// TIA Portal V17 export
// export: Created 2025-03-05T08:03:34.1256908Z, ExportSetting WithDefaults, DisplayName Totally Integrated Automation Portal, DisplayVersion V17 Update 8, DisplayName TIA Portal Openness, DisplayVersion V17 Update 8, DisplayName TIA Portal Version Control Interface, DisplayVersion V17, DisplayName SINAMICS Startdrive Advanced, DisplayVersion V17 SP2, DisplayName SINAMICS Startdrive G110M, G120, G120C, G120D, G120P, G115D, DisplayVersion V17 SP2, DisplayName SINAMICS Startdrive G130, G150, S120, S150, SINAMICS MV, S210, DisplayVersion V17 SP2, DisplayName STEP 7 Professional, DisplayVersion V17 Update 8, DisplayName SINUMERIK ONE STEP 7 Toolbox, DisplayVersion V17 Update 12, DisplayName SINUMERIK 840D sl STEP 7 Toolbox, DisplayVersion V17 Update 12, DisplayName STEP 7 Safety, DisplayVersion V17 Update 6, DisplayName WinCC Advanced, DisplayVersion V17 Update 8
DATA_BLOCK "DB22741_LOAD_FEEDER_TIME_SEQUENCE_HOPPER_3_UNIT_02"   // DB22741
{ DB_Accessible_From_OPC_UA := 'FALSE' }
VERSION : 0.1
// stored: AutoNumber false, DBAccessibleFromOPCUA false, DBAccessibleFromWebserver true, InstanceOfName FB22701_LOAD_FEEDER_SEQUENCE_TIME, InstanceOfType FB
"FB22701_LOAD_FEEDER_SEQUENCE_TIME"
   // VAR_INPUT
   //    iCONTROL_ON_DELAYED : Bool;
   //    iPNEUMATIC_FEEDBACK_ON : Bool;
   //    iFEEDER_PROFINET_MODE_ACTIVE_FAULT : Bool;
   //    iFEEDER_LINE_NOT_READY_FAULT : Bool;
   //    iMOTOR_STIRRER_CONDITIONS : Bool;
   //    iHOPPER_FEEDBACK_PRESSURE : Real;
   //    iHOPPER_MOTOR_STIRRER_FEEDBACK_SPEED : Real;
   //    iPOWDER_FEEDER_HOPPER_FEEDBACK_PRESSURE : Real;
   //    iTRANSFER_POWDER_VALVE_FEEDBACK_ON : Bool;
   //    iTRANSFER_POWDER_VALVE_FEEDBACK_OFF : Bool;
   //    iPOWDER_FLOW_ON : Bool;
   //    iSTART_MANUAL_REQUEST : Bool;
   //    iSTART_SEMI_REQUEST : Bool;
   //    iSTART_AUTO_REQUEST : Bool;
   //    iSTOP_MANUAL_REQUEST : Bool;
   //    iSTOP_SEMI_REQUEST : Bool;
   //    iSTOP_AUTO_REQUEST : Bool;
   // END_VAR
   // VAR_OUTPUT
   //    oEXCEEDED_TIME_ALARM : Bool;
   //    oOUT_OF_RANGE_ALARM : Bool;
   //    oLOST_CONDITIONS : Bool;
   //    oIS_ALARMS : Bool;
   // END_VAR
   // VAR_IN_OUT
   //    MOTOR_STIRRER_SETPOINT : DInt;
   //    PRESSURE_SETPOINT : Real;
   // END_VAR
   // VAR RETAIN
   //    DATA_SEQUENCE : "GENERAL_DATA_SEQUENCES";
   //    HMI_STANDARD : "HMI_DATA_START_STOP";
   //    INPUT_SETTINGS : Struct
   //       UNIT_NUMBER : Int := 2;
   //       HOPPER_NUMBER : Int := 3;
   //    END_STRUCT;
   //    HMI_SEQUENCE : Struct
   //       HMI_SEQUENCE_RUNNING : Bool;
   //       HMI_SEQUENCE_DONE : Bool;
   //       HMI_SET_TIME_LOAD : UDInt;
   //       HMI_MAX_ON_SET_TIME : UDInt;
   //       HMI_FEEDBACK_TIME_LOAD : Int;
   //       HMI_PRESSURE_INCREMENT : Real;
   //    END_STRUCT;
   //    ACTIONS_SEQUENCE : Struct
   //       REQ_START_TRANSFER_POWDER_VALVE : Bool;
   //       REQ_STOP_TRANSFER_POWDER_VALVE : Bool;
   //       REQ_START_PRESSURE_GAS_CONTROL : Bool;
   //       REQ_STOP_PRESSURE_GAS_CONTROL : Bool;
   //       REQ_START_PRESSURE_GAS_VALVE : Bool;
   //       REQ_STOP_PRESSURE_GAS_VALVE : Bool;
   //       REQ_START_RELIEF_GAS_VALVE : Bool;
   //       REQ_STOP_RELIEF_GAS_VALVE : Bool;
   //       SETPOINT_PRESSURE : Real;
   //       REQUEST_START_MOTOR_STIRRER : Bool;
   //       REQUEST_STOP_MOTOR_STIRRER : Bool;
   //       SETPOINT_MOTOR_STIRRER : DInt;
   //    END_STRUCT;
   //    CONTROL_SEQUENCE : Struct
   //       HOPPER_PRESSURE_IN_RANGE : Bool;
   //       HOPPER_MOTOR_STIRRER_IN_RANGE : Bool;
   //       HOPPER_STIRRER_LOW_RANGE : DInt;
   //       HOPPER_STIRRER_HIGH_RANGE : DInt;
   //       HOPPER_PRESSURE_LOW_RANGE : Real;
   //       HOPPER_PRESSURE_HIGH_RANGE : Real;
   //       HOPPER_PRESSURE_INCREMENT : Real;
   //       TIMER_IS_OVER : Bool;
   //       INITIAL_TIME_SET : DInt;
   //       TIMER_MATERIAL_APPLIED : Time;
   //    END_STRUCT;
   //    INTERNAL : Struct
   //       TRIGGER_RAISING_EDGE_1 : Bool;
   //       TRIGGER_RAISING_EDGE_2 : Bool;
   //       TRIGGER_RAISING_EDGE_3 : Bool;
   //    END_STRUCT;
   //    TIMERS : Struct
   //       TIMER_1 : TON_TIME;
   //       TIMER_2 : TON_TIME;
   //       TIMER_3 : TON_TIME;
   //       TIMER_4 : TON_TIME;
   //       TIMER_5 : TON_TIME;
   //       TIMER_6 : TON_TIME;
   //       TIMER_7 : TON_TIME;
   //       TIMER_8 : TON_TIME;
   //       TIMER_9 : TON_TIME;
   //       TIMER_10 : TON_TIME;
   //    END_STRUCT;
   // END_VAR
BEGIN
END_DATA_BLOCK
